# EPICS autosave request: ADADSC/iocs/adscIOC/iocBoot/iocAdsc/auto_settings.req
file "ADBase_settings.req", P=$(P),  R=det1:
file "adsc_settings.req",   P=$(P),  R=det1:
